(*
SPDX-FileCopyrightText: © 2026 Oleksandr Tiutyk <trofimich@gmail.com>
SPDX-License-Identifier: MIT
License: https://opensource.org/license/mit
*)

(*!
<summary>Deletes a file through cyclic task execution.</summary>
<description>
Use one owner task. Configure the path, target, path type and timeout before Start and keep them unchanged
until STOPPED. A missing path is rejected during execution; native errors propagate through Task failure
handling. There is no separate existence check and no conversion of a native not-found error to success.
Continue Execute through stopping, including after cancellation: an already submitted request is drained, not
rolled back. Failure or cancellation does not prove the file still exists. Reset preserves configuration.
</description>
*)

{attribute 'no_explicit_call' := 'do not call this function block directly'}
FUNCTION_BLOCK DeleteFile EXTENDS TOF_Tasks.Task IMPLEMENTS IFileSystemTask
VAR_STAT
	//! <summary>Static type metadata available before the base task initializes its default name.</summary>
	{attribute 'hide'}
	_ClassName : STRING := __POUNAME();
END_VAR
VAR
    _DeleteFile : Tc2_System.FB_FileDelete;
END_VAR

(*!
<summary>Selects the ADS target for the native filesystem operation.</summary>
<description>
Configure before Start and keep unchanged until STOPPED; the setter stores configuration without submitting
I/O.
</description>
*)
{attribute 'monitoring' := 'call'}
{attribute 'OPC.UA.DA.Property' := '1'}
{attribute 'OPC.UA.DA' := '1'}
PROPERTY AmsNetId : Tc2_System.T_AmsNetID
GET
AmsNetId := _DeleteFile.sNetId;
END_GET
SET
_DeleteFile.sNetId := AmsNetId;
END_SET
END_PROPERTY

(*!
<summary>Provides the concrete type name used in diagnostics.</summary>
<description>
Returns borrowed read-only metadata; keep the instance alive and do not modify the referenced string.
Initialized static storage is ready during base Task.FB_init; this getter has no side effects or exceptions.
</description>
*)
{attribute 'monitoring' := 'call'}
PROPERTY ClassName : REFERENCE TO STRING
GET
ClassName REF= _ClassName;
END_GET
END_PROPERTY

(*!
<summary>Provides the configured path for the file operation.</summary>
<description>
The setter copies text without performing I/O. Configure before Start and keep unchanged until STOPPED; Reset
preserves it. The native service determines whether the path is usable.
</description>
*)
{attribute 'monitoring' := 'call'}
{attribute 'OPC.UA.DA.Property' := '1'}
{attribute 'OPC.UA.DA' := '1'}
PROPERTY FilePath : Tc2_System.T_MaxString
GET
FilePath := _DeleteFile.sPathName;
END_GET
SET
_DeleteFile.sPathName := FilePath;
END_SET
END_PROPERTY

(*!
<summary>Provides the library namespace used in diagnostics.</summary>
<description>Returns borrowed read-only namespace storage; do not modify the referenced string.</description>
*)
{attribute 'monitoring' := 'call'}
PROPERTY NamespaceName : REFERENCE TO STRING
GET
NamespaceName REF= CurrentNamespace.Name;
END_GET
END_PROPERTY

(*!
<summary>Resets the native request edge after the task has stopped.</summary>
<description>
Preserves configured inputs and does not undo completed filesystem effects. Pending I/O must finish during
stopping before this hook runs.
</description>
*)
METHOD PROTECTED OnReset
_DeleteFile(bExecute := FALSE);
END_METHOD

(*!
<summary>Submits and advances native deletion of the configured file.</summary>
<description>
Validates required configuration before submitting the request. Native errors raise an exception for the base
Task failure/stopping path without dynamic string-builder allocations. Normal completion reports DONE only
after the native block is no longer busy. No rollback is performed.
</description>
<param name="processingState">BUSY while pending; DONE after native completion without an error.</param>
<param name="stopReasonMessage">Not changed here; failures are passed through exceptions.</param>
*)
METHOD PROTECTED OnRunning
VAR_OUTPUT
	processingState : TOF_Tasks.TASK_PROCESSING_STATE;
END_VAR
VAR_IN_OUT
	stopReasonMessage : TOF_Core.ERROR_MESSAGE;
END_VAR
VAR
	formattedExceptionMessage : TOF_Core.ERROR_MESSAGE;
END_VAR
IF NOT _DeleteFile.bExecute THEN 
	IF TOF_Core.Strings.IsNullOrWhiteSpace(stringToCheck := _DeleteFile.sPathName) THEN
		TOF_Core.Exceptions.ThrowDataMemberNotSpecified(
			sourceNamespaceName := NamespaceName,
			sourceClassName := ClassName,
			sourcePOUName := __POUNAME(),
			sourcePosition := __POSITION(),
			dataMemberName := 'FilePath'
		);		
	END_IF
END_IF

_DeleteFile(bExecute := TRUE);

IF _DeleteFile.bError THEN
	TOF_Core.WideStrings.Append255(
		formattedExceptionMessage,
		"An error occurred while deleting the file '",
		TO_WSTRING(_DeleteFile.sPathName),
		"'");

	FileSystemExceptions.ThrowFileSystem(
		sourceNamespaceName := NamespaceName,
		sourceClassName := ClassName,
		sourcePOUName := __POUNAME(),
		sourcePosition := __POSITION(),
		message := formattedExceptionMessage,
		errorCode := _DeleteFile.nErrId
	);
END_IF

IF NOT _DeleteFile.bBusy THEN
	processingState := TOF_Tasks.TASK_PROCESSING_STATE.DONE;
END_IF
END_METHOD

(*!
<summary>Waits for an already submitted operation before task termination.</summary>
<description>
Runs for every stop reason. Advances the pending FB with bExecute=FALSE without issuing another request.
Completion does not roll back side effects. Keep configuration and borrowed buffers valid until STOPPED.
</description>
<param name="readyToRelease">TRUE when the underlying FB is no longer busy.</param>
*)
METHOD PROTECTED OnStopping
VAR_OUTPUT
	readyToRelease : BOOL;
END_VAR
IF _DeleteFile.bBusy THEN
	_DeleteFile(bExecute := FALSE);
END_IF

readyToRelease := NOT _DeleteFile.bBusy;
END_METHOD

(*!
<summary>Selects the native path context for the filesystem request.</summary>
<description>
Configure before Start and keep unchanged until STOPPED. It is passed to the native operation, not used as a
path-validity result. Reset preserves it.
</description>
*)
{attribute 'monitoring' := 'call'}
{attribute 'OPC.UA.DA.Property' := '1'}
{attribute 'OPC.UA.DA' := '1'}
PROPERTY PathType : Tc2_System.E_OpenPath
GET
PathType := _DeleteFile.ePath;
END_GET
SET
_DeleteFile.ePath := PathType;
END_SET
END_PROPERTY

(*!
<summary>Reports the size of this concrete instance in bytes.</summary>
*)
{attribute 'monitoring' := 'call'}
PROPERTY SelfSize : ULINT
GET
SelfSize := XSIZEOF(THIS^);
END_GET
END_PROPERTY

(*!
<summary>Configures the timeout passed to native operation requests.</summary>
<description>
Set before Start and keep unchanged until STOPPED. Reset preserves this value. It is not an overall task
deadline or a guarantee of resource release after a timeout.
</description>
*)
{attribute 'monitoring' := 'call'}
{attribute 'OPC.UA.DA.Property' := '1'}
{attribute 'OPC.UA.DA' := '1'}
PROPERTY Timeout : TIME
GET
Timeout := _DeleteFile.tTimeout;
END_GET
SET
_DeleteFile.tTimeout := Timeout;
END_SET
END_PROPERTY

END_FUNCTION_BLOCK

(* stored: Version 1.1.0.1
   POU DeleteFile: Id {f7444039-d4c1-498f-9d80-3570b1d85b65}, SpecialFunc None
   Folder Inputs: Id {5c734593-9cb0-4d4a-a8bd-280e5f7cf47f}
   Folder Members to override: Id {8c98957e-0b2c-4bc7-ad6a-510d4f07ad24}
   Property AmsNetId: Id {51e41684-991f-4895-ae24-ce493fb5ef2c}
   Get Get: Id {76322297-0858-4421-a0f5-6bbdc5b131fb}
   Set Set: Id {745ae5f5-8fb5-4563-93fc-b37de88ffcb3}
   Property ClassName: Id {9a0868c1-10bc-4fb1-9326-3325da31a11b}
   Get Get: Id {7319f073-76e9-4be5-bd91-98627ec5b619}
   Property FilePath: Id {d92d06d0-9330-4ded-b02a-eb12d17df177}
   Get Get: Id {b4f03ed5-6f36-4301-ba38-819c4e9a9c6a}
   Set Set: Id {d40f0212-7cfd-4ab0-9944-711f5bbe86a1}
   Property NamespaceName: Id {6dbfdf1c-1abc-4260-b785-e313a600550a}
   Get Get: Id {e7b99e4c-8c32-4968-8443-d5548a868161}
   Method OnReset: Id {d1362757-d3ac-47a4-8843-3c884393e309}
   Method OnRunning: Id {94b4f428-70c7-4323-9b12-6f7c9f13f4aa}
   Method OnStopping: Id {1f9243b4-249b-4e10-a8ba-a9ada8bba94c}
   Property PathType: Id {04d5602f-b967-48be-8eee-fabfe0730217}
   Get Get: Id {0a70ed3a-ad22-4012-998e-cad8adb6f0ec}
   Set Set: Id {17f4d9e6-d7fb-441b-a237-6a68c55281e2}
   Property SelfSize: Id {b9e0f797-1600-4e2b-aeef-634d4ea22c0b}
   Get Get: Id {6ca5367a-528c-4d24-a82f-7f843c438268}
   Property Timeout: Id {bbee8d51-257c-48ae-bf00-0819c028fd98}
   Get Get: Id {b5e1ae9e-d6a8-42b3-9294-f0972e8a4b98}
   Set Set: Id {73b0fc19-215f-4912-8e36-2f185992f3be} *)
